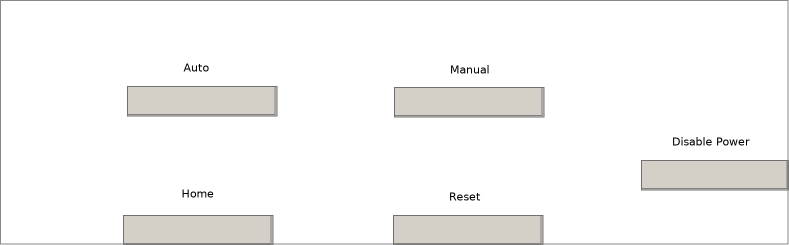
VISUALIZATION Visualization_1  // 789x245
    Button (127,86 150x30)
        tap MAIN.bUserStart
    Button (394,87 150x30)
        tap MAIN.bManual p1329445385=TRUE
    Label (390,182 150x30), "Reset"
    Button (393,215 150x30)
        tap MAIN.bReset
    Button (123,215 150x30)
        tap MAIN.bHome
    Label (123,53 150x30), "Auto"
    Label (123,179 150x30), "Home"
    Label (395,55 150x30), "Manual"
    Label (636,127 150x30), "Disable Power"
    Button (641,160 148x30)
        tap MAIN.bPowerDisable
END_VISUALIZATION

(* stored: Version 1.1.0.1, ProductVersion 3.1.4024.6
   Visu Visualization_1: Id {ab84306d-d93c-47e2-8082-5d935c879ad9} *)
